// TIA Portal V19 export
TYPE "LAF_typeUnitInterface"
TITLE = LAF_typeUnitInterface
// Interface structure of the unit
// stored: Access Published
   STRUCT
      information : "LAF_typeMachineInformation";
      status { ExternalWritable := 'False'} : "LAF_typeMachineStatus";
      enableControlInterfaces : "LAF_typeEnableControlInterfaces";   // Enable interfaces to control the unit
      controlModeStateManager : "LUC_typeManagerInterface";
      specialFunctions : "LAF_typeSpecialFunctions";   // Special functions of the current unit
      signalStack { ExternalWritable := 'False'} : "LUC_typeSignalStackByDWord";   // Signalstack
      alarms { ExternalWritable := 'False'} : "LAF_typeAlarms";   // Alarms inside the unit
      currentMode { ExternalWritable := 'False'} : String;   // Current mode as a string
      currentState { ExternalWritable := 'False'} : String;   // Current state as a string
      history { ExternalWritable := 'False'} : Array[0..15] of "LUC_typeModeState";
      modeStateTimeStatistics { ExternalWritable := 'False'} : "LUC_typeUnitModeStateTimes";
   END_STRUCT;
   // // history[0] : Current mode and state. In this case, duration stores the starttime, not the duration, you can ignore it.
END_TYPE
